(* IEC 61131-3 sources: AXOpen/src/core/app/src, 3 files *)

(* ---- recipe.st ---- *)
{#ix-attr:[Container(Layout.Tabs)]}
{#ix-attr:[Group(GroupLayout.GroupBox)]}
{#ix-set:AttributeName = "This is some structure"}
CLASS PUBLIC Recipe
    VAR PUBLIC
        Header : ReciepeHeader;
        Measurements : Measurements;
        Colors : Colors;
    END_VAR
END_CLASS

TYPE
    Colors : (RED, GREEN, BLUE);
END_TYPE

{#ix-attr:[Container(Layout.Stack)]}
CLASS PUBLIC ReciepeHeader
    VAR PUBLIC
        Name : STRING;
    END_VAR
END_CLASS

{#ix-attr:[Container(Layout.Tabs)]}
CLASS PUBLIC Measurements
    VAR PUBLIC
        {#ix-set:AttributeName = "Dimension X"}
        DimX : ContinuesValueCheckData;
        {#ix-set:AttributeName = "Dimension Y"}
        DimY : ContinuesValueCheckData;
        {#ix-set:AttributeName = "Dimension Z"}
        DimZ : ContinuesValueCheckData;
        {#ix-set:AttributeName = "Inside temp °C"}
        TemperatureIn : ContinuesValueCheckData;
        {#ix-set:AttributeName = "Outside temp °C"}
        TemperatureOut : ContinuesValueCheckData;
    END_VAR
END_CLASS

{#ix-attr:[Container(Layout.Wrap)]}
{#ix-attr:[Group(GroupLayout.GroupBox)]}
CLASS PUBLIC ContinuesValueCheckData
    VAR PUBLIC
        Min : REAL;
        Measured : REAL;
        Max : REAL;
    END_VAR
END_CLASS

(* ---- configuration.st ---- *)
USING VmT;
CONFIGURATION MyConfiguration
    TASK Main(Interval := T#10ms, Priority := 1);
    PROGRAM P1 WITH Main: MyProgram;
    PROGRAM P2 WITH Main: ProgramExample;

    VAR_GLOBAL
        {S7.extern=ReadWrite}
        Recipe : Recipe;
        {#ix-set:AttributeName = "If counting PLC is alive"}
        {S7.extern=ReadWrite}
        I_am_alive : ULINT;
        {S7.extern=ReadWrite}
        AxoSequencers : AxoSequencerExamples.SequencerExample;
        {S7.extern=ReadWrite}
        AxoSequencerContainer : AxoSequencerContainerExamples.SequencerContainerExample;
        {S7.extern=ReadWrite}
        AxoTasks : AxoTaskExamples.Tasks;
        {S7.extern=ReadWrite}
        AxoTaskDocu : AxoTaskExamples.AxoTaskDocuExample;
        {S7.extern=ReadWrite}
        myComponentExample : AxoComponentExamples.ComponentExampleContext;
        {S7.extern=ReadWrite}
        myComponentHeaderOnlyExample : AxoComponentExamples.ComponentHeaderOnlyExampleContext;
        {S7.extern=ReadWrite}
        AxoRemoteTasks : AxoRemoteTaskExamples.RemoteTasks;
        {S7.extern=ReadWrite}
        AxoToggleTasks : AxoToggleTaskExamples.Tasks;
        {S7.extern=ReadWrite}
        AxoToggleTaskDocu : AxoToggleTaskExamples.AxoToggleTaskDocuExample;
        {S7.extern=ReadWrite}
        AxoMomentaryTasks : AxoMomentaryTaskExamples.Tasks;
        {S7.extern=ReadWrite}
        AxoMomentaryTaskDocu : AxoMomentaryTaskExamples.AxoMomentaryTaskDocuExample;
        {S7.extern=ReadWrite}
        AxoMessengers : AxoStaticMessengerExample.Messengers;
        {S7.extern=ReadWrite}
        AxoMessengersDocu : AxoStaticMessengerDocuExample.Messengers;
        {S7.extern=ReadWrite}
        AxoRtc : AxoRtc.AxoS71500Rtc;
        {S7.extern=ReadWrite}
        AxoTextListExampleContext : AxoTextListExample.AxoTextListExampleContext;
        {S7.extern=ReadWrite}
        AxoByteArrayExampleContext : AxoByteArrayExample.AxoByteArrayExampleContext;
        {S7.extern=ReadWrite}
        AxoBoolArrayExampleContext : AxoBoolArrayExample.AxoBoolArrayExampleContext;
        {S7.extern=ReadWrite}
        AxoLoggers : AxoLoggerExamples.Loggers;
        {S7.extern=ReadWrite}
        D_111 : AxoDialogExamples.Dialogs;
        {S7.extern=ReadWrite}
        D_222 : AxoDialogExamples.Dialogs;
        // Issues
        {S7.extern=ReadWrite}
        gh_ptku_8 : Layouts.Tabbed.weather;

        {S7.extern=ReadWrite}
        AxoS71500Rtc : AxoS71500RtcContext;

        {S7.extern=ReadWrite}
        Simatic1500Alarming : Simatic1500AlarmingContext;

    END_VAR
END_CONFIGURATION

(* ---- program.st ---- *)
USING AXOpen.Core;

PROGRAM MyProgram
    VAR_EXTERNAL
        I_am_alive : ULINT;
        AxoSequencers : AxoSequencerExamples.SequencerExample;
        AxoSequencerContainer : AxoSequencerContainerExamples.SequencerContainerExample;
        AxoTasks : AxoTaskExamples.Tasks;
        AxoTaskDocu : AxoTaskExamples.AxoTaskDocuExample;
        myComponentExample : AxoComponentExamples.ComponentExampleContext;
        myComponentHeaderOnlyExample : AxoComponentExamples.ComponentHeaderOnlyExampleContext;
        AxoRemoteTasks : AxoRemoteTaskExamples.RemoteTasks;
        AxoToggleTasks : AxoToggleTaskExamples.Tasks;
        AxoToggleTaskDocu : AxoToggleTaskExamples.AxoToggleTaskDocuExample;
        AxoMomentaryTasks : AxoMomentaryTaskExamples.Tasks;
        AxoMomentaryTaskDocu : AxoMomentaryTaskExamples.AxoMomentaryTaskDocuExample;
        AxoMessengers : AxoStaticMessengerExample.Messengers;
        AxoMessengersDocu : AxoStaticMessengerDocuExample.Messengers;
        AxoTextListExampleContext : AxoTextListExample.AxoTextListExampleContext;
        AxoByteArrayExampleContext : AxoByteArrayExample.AxoByteArrayExampleContext;
        AxoBoolArrayExampleContext : AxoBoolArrayExample.AxoBoolArrayExampleContext;
        AxoLoggers : AxoLoggerExamples.Loggers;
        D_111 : AxoDialogExamples.Dialogs;
        D_222 : AxoDialogExamples.Dialogs;
        //Dialogs : AxoDialogExamples.Dialogs;
        AxoRtc : AxoRtc.AxoS71500Rtc;
        AxoS71500Rtc : AxoS71500RtcContext;
        Simatic1500Alarming : Simatic1500AlarmingContext;
    END_VAR

    I_am_alive := I_am_alive + ULINT#1;

    AxoTasks.Run();
    AxoTaskDocu.Run();
    AxoToggleTasks.Run();
    AxoToggleTaskDocu.Run();
    AxoSequencers.Run();
    AxoSequencerContainer.Run();
    myComponentExample.Run();
    myComponentHeaderOnlyExample.Run();
    AxoRemoteTasks.Run();
    AxoMomentaryTasks.Run();
    AxoMomentaryTaskDocu.Run();

    AxoMessengers.Run();
    AxoMessengers.InjectRtc(AxoRtc);
    AxoMessengersDocu.Run();
    AxoMessengersDocu.InjectRtc(AxoRtc);
    AxoTextListExampleContext.Run();

    AxoByteArrayExampleContext.Run();
    AxoBoolArrayExampleContext.Run();

    AxoLoggers.InjectRtc(AxoRtc);
    AxoLoggers.Run();

    D_111.InjectRtc(AxoRtc);
    D_111.Run();

    D_222.InjectRtc(AxoRtc);
    D_222.Run();

    AxoS71500Rtc.Run();

    Simatic1500Alarming.Run();

END_PROGRAM
